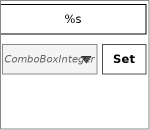
VISUALIZATION vAxisBrakeControl  // 150x130
VAR_IN_OUT
	fbData	: fb_ServoAxis;
END_VAR
    Rectangle (102,44 44x30), "Set", colour toggle: fbData.bSetNewBrakeCtrl, input disabled if: fbData.iWorkStep_Axis <>15
        toggle fbData.bSetNewBrakeCtrl p2164770859=TRUE
    Rectangle (0,4 146x30), "%s", text variable: TO_STRING(fbData.nAct_BrakeMode)
    ComboBoxInteger (2,44 95x30), variable: fbData.nNew_BrakeMode, input disabled if: fbData.iWorkStep_Axis <>15
END_VISUALIZATION

(* stored: Version 1.1.0.1, ProductVersion 3.1.4024.15
   Visu vAxisBrakeControl: Id {20858d17-42b9-4fc9-b3d1-223aee237698} *)
